// TIA Portal V20 export
FUNCTION_BLOCK "LER_StackLight"   // FB8, LAD
// stored: Access Published, MemoryReserve 100, SetENOAutomatically false
   VAR_INPUT
      stateDetail : "LER_typeStateDetail";
      powerOn : Bool;
      auto : Bool;
      manual : Bool;
   END_VAR
   VAR_OUTPUT
      setDone : Bool;
      signalStack : "LUC_typeSignalStackConfiguration";
   END_VAR
   VAR
      statExcute : Bool;
      statDefault : Bool;
      statReset : Bool;
      statResetDone : Bool;
      statPreStateDetail : "LER_typeStateDetail";
   END_VAR
   VAR_TEMP
      signalStackDelete : "LUC_typeSignalStackConfiguration";
      tempRetVal : Array[0..9] of Int;
   END_VAR
   VAR_TEMP   // added for the SCL form of the ladder/FBD networks
      _w1 : Bool;
   END_VAR
BEGIN

REGION Network 1 (SCL): stateDefault
   // stateDetail is All False
   IF (#stateDetail."Turn off" OR #stateDetail."Technical issue or alarm" OR #stateDetail."Internal starved" OR #stateDetail."Emergency or hazardous stop" OR #stateDetail.Overheat OR #stateDetail.Warning OR
       #stateDetail."External starved or blocked" OR #stateDetail."QC required soon" OR #stateDetail."Controlled Stop" OR #stateDetail."Ready to start" OR #stateDetail."Producing(running)") = 0 THEN
       #statDefault := TRUE;
       #statExcute := TRUE;
   END_IF;
END_REGION

REGION Network 2: reset
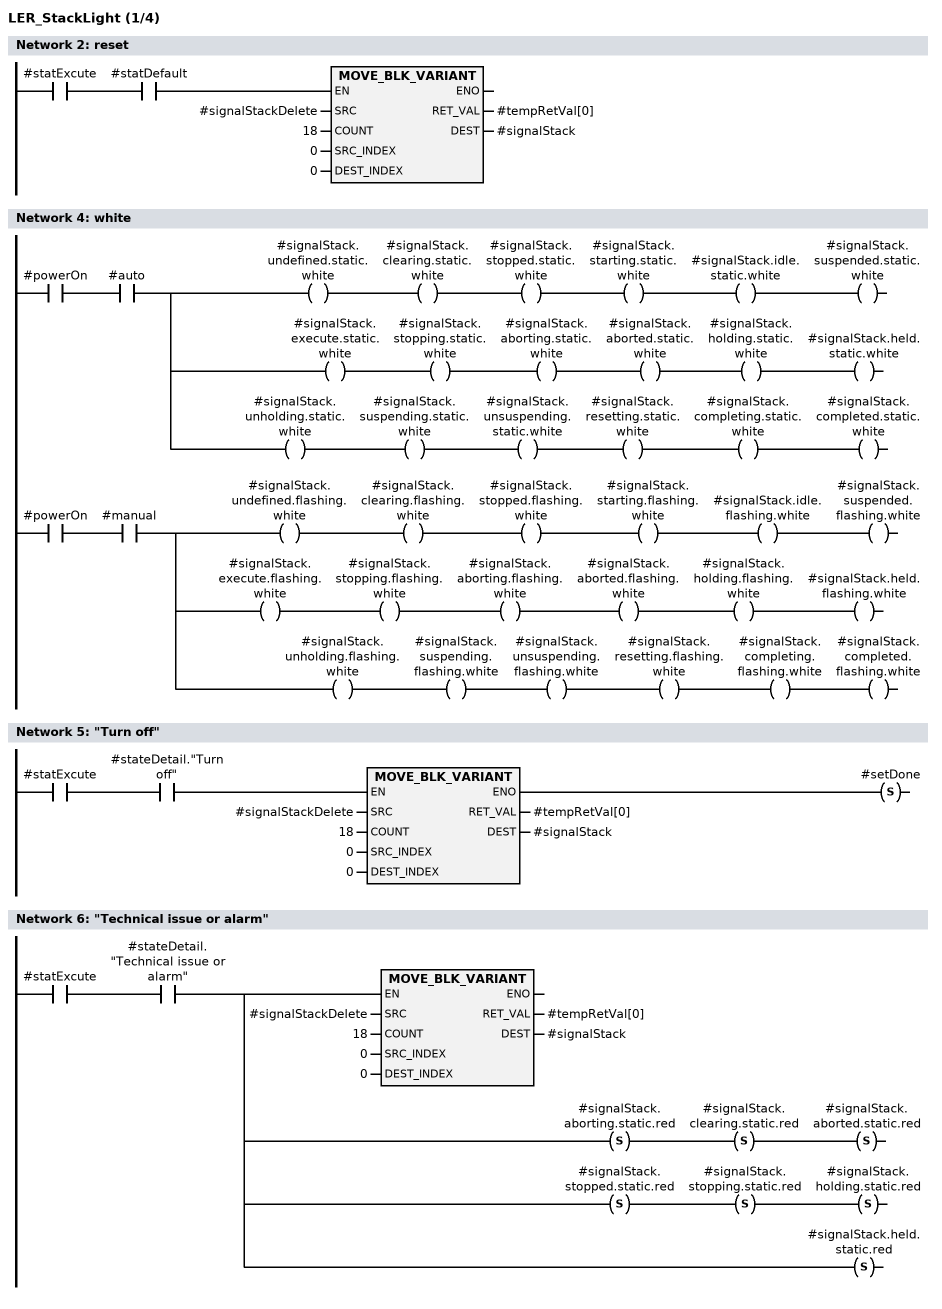
   RUNG wire#powerrail
      Contact( #statExcute )
      Contact( #statDefault )
      MOVE_BLK_VARIANT(SRC := #signalStackDelete, COUNT := 18, SRC_INDEX := 0, DEST_INDEX := 0, Ret_Val => #tempRetVal[0], DEST => #signalStack)
   END_RUNG
   // the same network as SCL:
   IF #statExcute AND #statDefault THEN
       #tempRetVal[0] := MOVE_BLK_VARIANT(SRC := #signalStackDelete,
                               COUNT := 18,
                               SRC_INDEX := 0,
                               DEST_INDEX := 0,
                               DEST => #signalStack);
   END_IF;
END_REGION

REGION Network 3 (SCL)
   IF #statPreStateDetail <> #stateDetail THEN
       #statExcute := TRUE;
       #statPreStateDetail := #stateDetail;
   END_IF;
END_REGION

REGION Network 4: white
   RUNG wire#powerrail
      Contact( #powerOn )
      Contact( #auto )
      wire#w1
      Coil( #signalStack.undefined.static.white )
      Coil( #signalStack.clearing.static.white )
      Coil( #signalStack.stopped.static.white )
      Coil( #signalStack.starting.static.white )
      Coil( #signalStack.idle.static.white )
      Coil( #signalStack.suspended.static.white )
   END_RUNG
   RUNG wire#w1
      Coil( #signalStack.execute.static.white )
      Coil( #signalStack.stopping.static.white )
      Coil( #signalStack.aborting.static.white )
      Coil( #signalStack.aborted.static.white )
      Coil( #signalStack.holding.static.white )
      Coil( #signalStack.held.static.white )
   END_RUNG
   RUNG wire#w1
      Coil( #signalStack.unholding.static.white )
      Coil( #signalStack.suspending.static.white )
      Coil( #signalStack.unsuspending.static.white )
      Coil( #signalStack.resetting.static.white )
      Coil( #signalStack.completing.static.white )
      Coil( #signalStack.completed.static.white )
   END_RUNG
   RUNG wire#powerrail
      Contact( #powerOn )
      Contact( #manual )
      wire#w2
      Coil( #signalStack.undefined.flashing.white )
      Coil( #signalStack.clearing.flashing.white )
      Coil( #signalStack.stopped.flashing.white )
      Coil( #signalStack.starting.flashing.white )
      Coil( #signalStack.idle.flashing.white )
      Coil( #signalStack.suspended.flashing.white )
   END_RUNG
   RUNG wire#w2
      Coil( #signalStack.execute.flashing.white )
      Coil( #signalStack.stopping.flashing.white )
      Coil( #signalStack.aborting.flashing.white )
      Coil( #signalStack.aborted.flashing.white )
      Coil( #signalStack.holding.flashing.white )
      Coil( #signalStack.held.flashing.white )
   END_RUNG
   RUNG wire#w2
      Coil( #signalStack.unholding.flashing.white )
      Coil( #signalStack.suspending.flashing.white )
      Coil( #signalStack.unsuspending.flashing.white )
      Coil( #signalStack.resetting.flashing.white )
      Coil( #signalStack.completing.flashing.white )
      Coil( #signalStack.completed.flashing.white )
   END_RUNG
   // the same network as SCL:
   #signalStack.undefined.static.white := #powerOn AND #auto;
   #signalStack.clearing.static.white := #signalStack.undefined.static.white;
   #signalStack.stopped.static.white := #signalStack.undefined.static.white;
   #signalStack.starting.static.white := #signalStack.undefined.static.white;
   #signalStack.idle.static.white := #signalStack.undefined.static.white;
   #signalStack.suspended.static.white := #signalStack.undefined.static.white;
   #signalStack.execute.static.white := #signalStack.undefined.static.white;
   #signalStack.stopping.static.white := #signalStack.undefined.static.white;
   #signalStack.aborting.static.white := #signalStack.undefined.static.white;
   #signalStack.aborted.static.white := #signalStack.undefined.static.white;
   #signalStack.holding.static.white := #signalStack.undefined.static.white;
   #signalStack.held.static.white := #signalStack.undefined.static.white;
   #signalStack.unholding.static.white := #signalStack.undefined.static.white;
   #signalStack.suspending.static.white := #signalStack.undefined.static.white;
   #signalStack.unsuspending.static.white := #signalStack.undefined.static.white;
   #signalStack.resetting.static.white := #signalStack.undefined.static.white;
   #signalStack.completing.static.white := #signalStack.undefined.static.white;
   #signalStack.completed.static.white := #signalStack.undefined.static.white;
   #signalStack.undefined.flashing.white := #powerOn AND #manual;
   #signalStack.clearing.flashing.white := #signalStack.undefined.flashing.white;
   #signalStack.stopped.flashing.white := #signalStack.undefined.flashing.white;
   #signalStack.starting.flashing.white := #signalStack.undefined.flashing.white;
   #signalStack.idle.flashing.white := #signalStack.undefined.flashing.white;
   #signalStack.suspended.flashing.white := #signalStack.undefined.flashing.white;
   #signalStack.execute.flashing.white := #signalStack.undefined.flashing.white;
   #signalStack.stopping.flashing.white := #signalStack.undefined.flashing.white;
   #signalStack.aborting.flashing.white := #signalStack.undefined.flashing.white;
   #signalStack.aborted.flashing.white := #signalStack.undefined.flashing.white;
   #signalStack.holding.flashing.white := #signalStack.undefined.flashing.white;
   #signalStack.held.flashing.white := #signalStack.undefined.flashing.white;
   #signalStack.unholding.flashing.white := #signalStack.undefined.flashing.white;
   #signalStack.suspending.flashing.white := #signalStack.undefined.flashing.white;
   #signalStack.unsuspending.flashing.white := #signalStack.undefined.flashing.white;
   #signalStack.resetting.flashing.white := #signalStack.undefined.flashing.white;
   #signalStack.completing.flashing.white := #signalStack.undefined.flashing.white;
   #signalStack.completed.flashing.white := #signalStack.undefined.flashing.white;
END_REGION

REGION Network 5: "Turn off"
   RUNG wire#powerrail
      Contact( #statExcute )
      Contact( #stateDetail."Turn off" )
      MOVE_BLK_VARIANT(SRC := #signalStackDelete, COUNT := 18, SRC_INDEX := 0, DEST_INDEX := 0, Ret_Val => #tempRetVal[0], DEST => #signalStack)
      S_Coil( #setDone )
   END_RUNG
   // the same network as SCL:
   #tempRetVal[0] := MOVE_BLK_VARIANT(EN := #statExcute AND #stateDetail."Turn off",
                           SRC := #signalStackDelete,
                           COUNT := 18,
                           SRC_INDEX := 0,
                           DEST_INDEX := 0,
                           DEST => #signalStack,
                           ENO => #_w1);
   IF #_w1 THEN #setDone := TRUE; END_IF;
END_REGION

REGION Network 6: "Technical issue or alarm"
   RUNG wire#powerrail
      Contact( #statExcute )
      Contact( #stateDetail."Technical issue or alarm" )
      wire#w1
      MOVE_BLK_VARIANT(SRC := #signalStackDelete, COUNT := 18, SRC_INDEX := 0, DEST_INDEX := 0, Ret_Val => #tempRetVal[0], DEST => #signalStack)
   END_RUNG
   RUNG wire#w1
      S_Coil( #signalStack.aborting.static.red )
      S_Coil( #signalStack.clearing.static.red )
      S_Coil( #signalStack.aborted.static.red )
   END_RUNG
   RUNG wire#w1
      S_Coil( #signalStack.stopped.static.red )
      S_Coil( #signalStack.stopping.static.red )
      S_Coil( #signalStack.holding.static.red )
   END_RUNG
   RUNG wire#w1
      S_Coil( #signalStack.held.static.red )
   END_RUNG
   // the same network as SCL:
   IF #statExcute AND #stateDetail."Technical issue or alarm" THEN
       #tempRetVal[0] := MOVE_BLK_VARIANT(SRC := #signalStackDelete,
                               COUNT := 18,
                               SRC_INDEX := 0,
                               DEST_INDEX := 0,
                               DEST => #signalStack);
       #signalStack.aborting.static.red := TRUE;
       #signalStack.clearing.static.red := TRUE;
       #signalStack.aborted.static.red := TRUE;
       #signalStack.stopped.static.red := TRUE;
       #signalStack.stopping.static.red := TRUE;
       #signalStack.holding.static.red := TRUE;
       #signalStack.held.static.red := TRUE;
   END_IF;
END_REGION

REGION Network 7: "Internal starved"
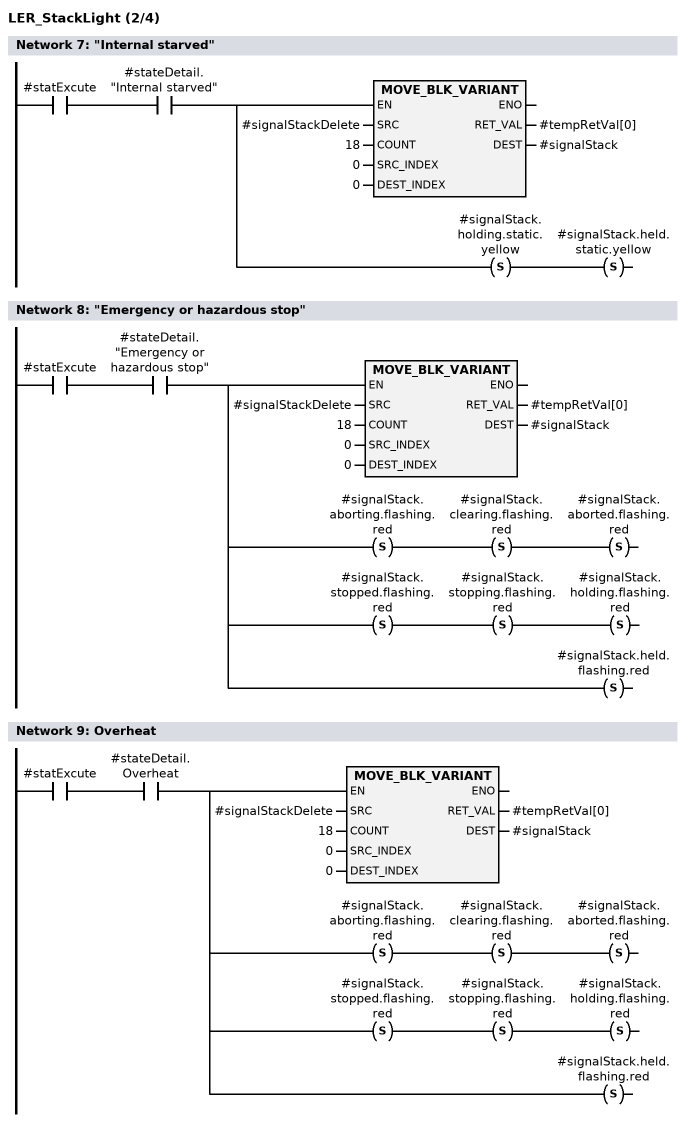
   RUNG wire#powerrail
      Contact( #statExcute )
      Contact( #stateDetail."Internal starved" )
      wire#w1
      MOVE_BLK_VARIANT(SRC := #signalStackDelete, COUNT := 18, SRC_INDEX := 0, DEST_INDEX := 0, Ret_Val => #tempRetVal[0], DEST => #signalStack)
   END_RUNG
   RUNG wire#w1
      S_Coil( #signalStack.holding.static.yellow )
      S_Coil( #signalStack.held.static.yellow )
   END_RUNG
   // the same network as SCL:
   IF #statExcute AND #stateDetail."Internal starved" THEN
       #tempRetVal[0] := MOVE_BLK_VARIANT(SRC := #signalStackDelete,
                               COUNT := 18,
                               SRC_INDEX := 0,
                               DEST_INDEX := 0,
                               DEST => #signalStack);
       #signalStack.holding.static.yellow := TRUE;
       #signalStack.held.static.yellow := TRUE;
   END_IF;
END_REGION

REGION Network 8: "Emergency or hazardous stop"
   RUNG wire#powerrail
      Contact( #statExcute )
      Contact( #stateDetail."Emergency or hazardous stop" )
      wire#w1
      MOVE_BLK_VARIANT(SRC := #signalStackDelete, COUNT := 18, SRC_INDEX := 0, DEST_INDEX := 0, Ret_Val => #tempRetVal[0], DEST => #signalStack)
   END_RUNG
   RUNG wire#w1
      S_Coil( #signalStack.aborting.flashing.red )
      S_Coil( #signalStack.clearing.flashing.red )
      S_Coil( #signalStack.aborted.flashing.red )
   END_RUNG
   RUNG wire#w1
      S_Coil( #signalStack.stopped.flashing.red )
      S_Coil( #signalStack.stopping.flashing.red )
      S_Coil( #signalStack.holding.flashing.red )
   END_RUNG
   RUNG wire#w1
      S_Coil( #signalStack.held.flashing.red )
   END_RUNG
   // the same network as SCL:
   IF #statExcute AND #stateDetail."Emergency or hazardous stop" THEN
       #tempRetVal[0] := MOVE_BLK_VARIANT(SRC := #signalStackDelete,
                               COUNT := 18,
                               SRC_INDEX := 0,
                               DEST_INDEX := 0,
                               DEST => #signalStack);
       #signalStack.aborting.flashing.red := TRUE;
       #signalStack.clearing.flashing.red := TRUE;
       #signalStack.aborted.flashing.red := TRUE;
       #signalStack.stopped.flashing.red := TRUE;
       #signalStack.stopping.flashing.red := TRUE;
       #signalStack.holding.flashing.red := TRUE;
       #signalStack.held.flashing.red := TRUE;
   END_IF;
END_REGION

REGION Network 9: Overheat
   RUNG wire#powerrail
      Contact( #statExcute )
      Contact( #stateDetail.Overheat )
      wire#w1
      MOVE_BLK_VARIANT(SRC := #signalStackDelete, COUNT := 18, SRC_INDEX := 0, DEST_INDEX := 0, Ret_Val => #tempRetVal[0], DEST => #signalStack)
   END_RUNG
   RUNG wire#w1
      S_Coil( #signalStack.aborting.flashing.red )
      S_Coil( #signalStack.clearing.flashing.red )
      S_Coil( #signalStack.aborted.flashing.red )
   END_RUNG
   RUNG wire#w1
      S_Coil( #signalStack.stopped.flashing.red )
      S_Coil( #signalStack.stopping.flashing.red )
      S_Coil( #signalStack.holding.flashing.red )
   END_RUNG
   RUNG wire#w1
      S_Coil( #signalStack.held.flashing.red )
   END_RUNG
   // the same network as SCL:
   IF #statExcute AND #stateDetail.Overheat THEN
       #tempRetVal[0] := MOVE_BLK_VARIANT(SRC := #signalStackDelete,
                               COUNT := 18,
                               SRC_INDEX := 0,
                               DEST_INDEX := 0,
                               DEST => #signalStack);
       #signalStack.aborting.flashing.red := TRUE;
       #signalStack.clearing.flashing.red := TRUE;
       #signalStack.aborted.flashing.red := TRUE;
       #signalStack.stopped.flashing.red := TRUE;
       #signalStack.stopping.flashing.red := TRUE;
       #signalStack.holding.flashing.red := TRUE;
       #signalStack.held.flashing.red := TRUE;
   END_IF;
END_REGION

REGION Network 10: Warning
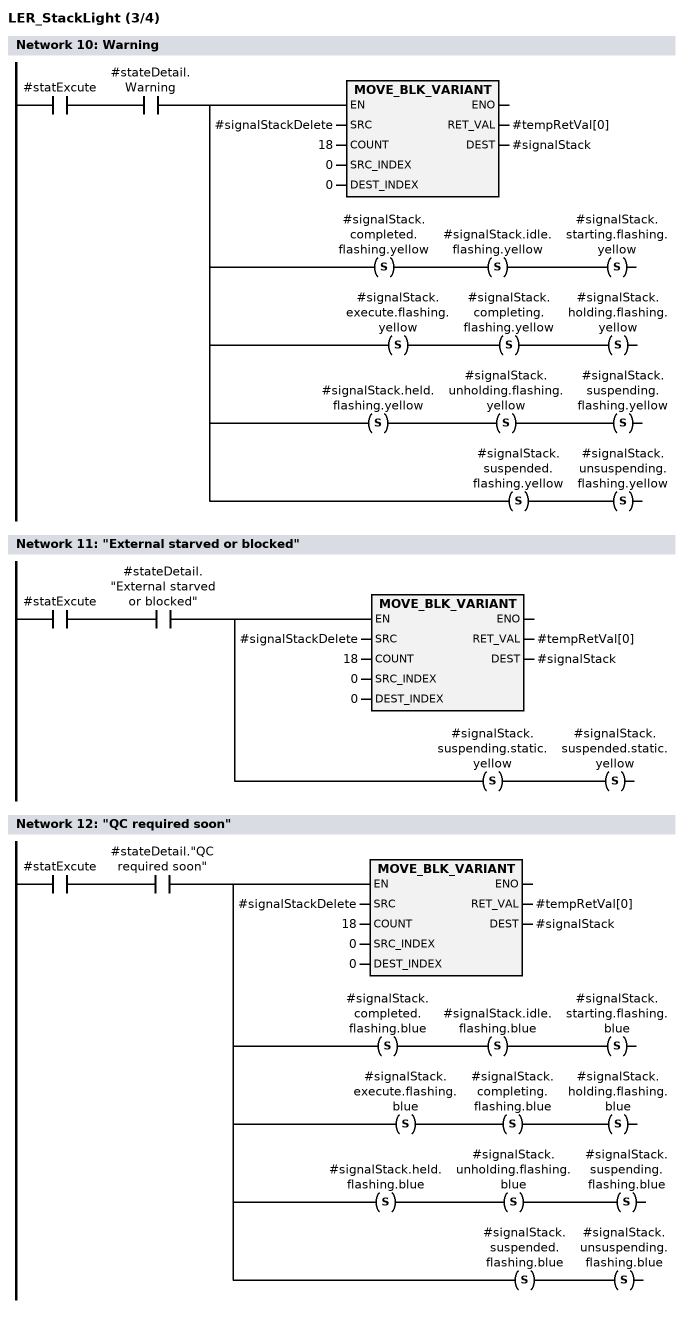
   RUNG wire#powerrail
      Contact( #statExcute )
      Contact( #stateDetail.Warning )
      wire#w1
      MOVE_BLK_VARIANT(SRC := #signalStackDelete, COUNT := 18, SRC_INDEX := 0, DEST_INDEX := 0, Ret_Val => #tempRetVal[0], DEST => #signalStack)
   END_RUNG
   RUNG wire#w1
      S_Coil( #signalStack.completed.flashing.yellow )
      S_Coil( #signalStack.idle.flashing.yellow )
      S_Coil( #signalStack.starting.flashing.yellow )
   END_RUNG
   RUNG wire#w1
      S_Coil( #signalStack.execute.flashing.yellow )
      S_Coil( #signalStack.completing.flashing.yellow )
      S_Coil( #signalStack.holding.flashing.yellow )
   END_RUNG
   RUNG wire#w1
      S_Coil( #signalStack.held.flashing.yellow )
      S_Coil( #signalStack.unholding.flashing.yellow )
      S_Coil( #signalStack.suspending.flashing.yellow )
   END_RUNG
   RUNG wire#w1
      S_Coil( #signalStack.suspended.flashing.yellow )
      S_Coil( #signalStack.unsuspending.flashing.yellow )
   END_RUNG
   // the same network as SCL:
   IF #statExcute AND #stateDetail.Warning THEN
       #tempRetVal[0] := MOVE_BLK_VARIANT(SRC := #signalStackDelete,
                               COUNT := 18,
                               SRC_INDEX := 0,
                               DEST_INDEX := 0,
                               DEST => #signalStack);
       #signalStack.completed.flashing.yellow := TRUE;
       #signalStack.idle.flashing.yellow := TRUE;
       #signalStack.starting.flashing.yellow := TRUE;
       #signalStack.execute.flashing.yellow := TRUE;
       #signalStack.completing.flashing.yellow := TRUE;
       #signalStack.holding.flashing.yellow := TRUE;
       #signalStack.held.flashing.yellow := TRUE;
       #signalStack.unholding.flashing.yellow := TRUE;
       #signalStack.suspending.flashing.yellow := TRUE;
       #signalStack.suspended.flashing.yellow := TRUE;
       #signalStack.unsuspending.flashing.yellow := TRUE;
   END_IF;
END_REGION

REGION Network 11: "External starved or blocked"
   RUNG wire#powerrail
      Contact( #statExcute )
      Contact( #stateDetail."External starved or blocked" )
      wire#w1
      MOVE_BLK_VARIANT(SRC := #signalStackDelete, COUNT := 18, SRC_INDEX := 0, DEST_INDEX := 0, Ret_Val => #tempRetVal[0], DEST => #signalStack)
   END_RUNG
   RUNG wire#w1
      S_Coil( #signalStack.suspending.static.yellow )
      S_Coil( #signalStack.suspended.static.yellow )
   END_RUNG
   // the same network as SCL:
   IF #statExcute AND #stateDetail."External starved or blocked" THEN
       #tempRetVal[0] := MOVE_BLK_VARIANT(SRC := #signalStackDelete,
                               COUNT := 18,
                               SRC_INDEX := 0,
                               DEST_INDEX := 0,
                               DEST => #signalStack);
       #signalStack.suspending.static.yellow := TRUE;
       #signalStack.suspended.static.yellow := TRUE;
   END_IF;
END_REGION

REGION Network 12: "QC required soon"
   RUNG wire#powerrail
      Contact( #statExcute )
      Contact( #stateDetail."QC required soon" )
      wire#w1
      MOVE_BLK_VARIANT(SRC := #signalStackDelete, COUNT := 18, SRC_INDEX := 0, DEST_INDEX := 0, Ret_Val => #tempRetVal[0], DEST => #signalStack)
   END_RUNG
   RUNG wire#w1
      S_Coil( #signalStack.completed.flashing.blue )
      S_Coil( #signalStack.idle.flashing.blue )
      S_Coil( #signalStack.starting.flashing.blue )
   END_RUNG
   RUNG wire#w1
      S_Coil( #signalStack.execute.flashing.blue )
      S_Coil( #signalStack.completing.flashing.blue )
      S_Coil( #signalStack.holding.flashing.blue )
   END_RUNG
   RUNG wire#w1
      S_Coil( #signalStack.held.flashing.blue )
      S_Coil( #signalStack.unholding.flashing.blue )
      S_Coil( #signalStack.suspending.flashing.blue )
   END_RUNG
   RUNG wire#w1
      S_Coil( #signalStack.suspended.flashing.blue )
      S_Coil( #signalStack.unsuspending.flashing.blue )
   END_RUNG
   // the same network as SCL:
   IF #statExcute AND #stateDetail."QC required soon" THEN
       #tempRetVal[0] := MOVE_BLK_VARIANT(SRC := #signalStackDelete,
                               COUNT := 18,
                               SRC_INDEX := 0,
                               DEST_INDEX := 0,
                               DEST => #signalStack);
       #signalStack.completed.flashing.blue := TRUE;
       #signalStack.idle.flashing.blue := TRUE;
       #signalStack.starting.flashing.blue := TRUE;
       #signalStack.execute.flashing.blue := TRUE;
       #signalStack.completing.flashing.blue := TRUE;
       #signalStack.holding.flashing.blue := TRUE;
       #signalStack.held.flashing.blue := TRUE;
       #signalStack.unholding.flashing.blue := TRUE;
       #signalStack.suspending.flashing.blue := TRUE;
       #signalStack.suspended.flashing.blue := TRUE;
       #signalStack.unsuspending.flashing.blue := TRUE;
   END_IF;
END_REGION

REGION Network 13: "Controlled Stop"
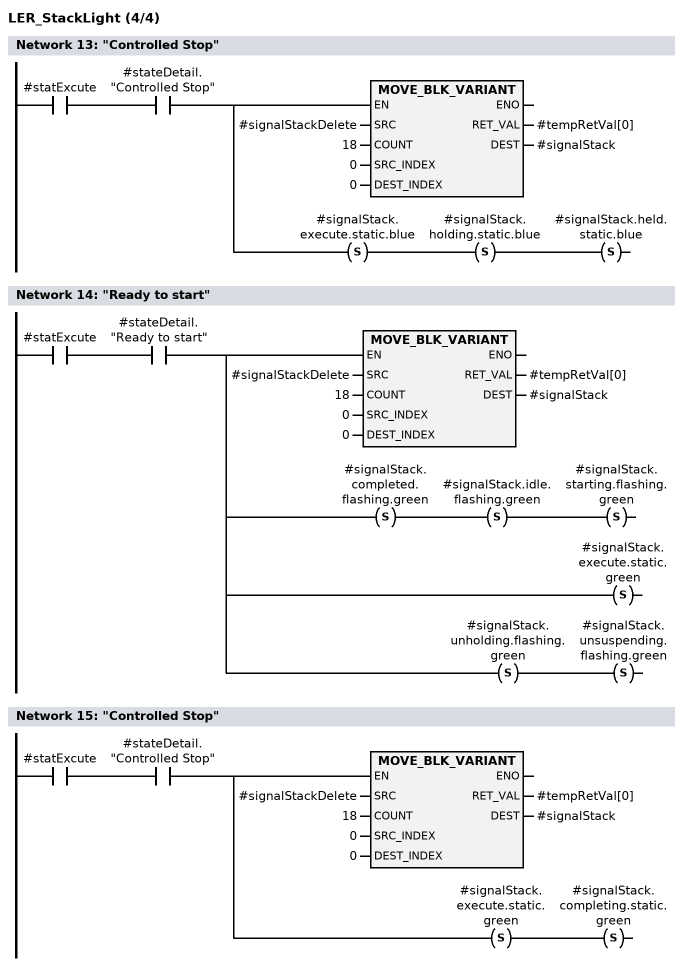
   RUNG wire#powerrail
      Contact( #statExcute )
      Contact( #stateDetail."Controlled Stop" )
      wire#w1
      MOVE_BLK_VARIANT(SRC := #signalStackDelete, COUNT := 18, SRC_INDEX := 0, DEST_INDEX := 0, Ret_Val => #tempRetVal[0], DEST => #signalStack)
   END_RUNG
   RUNG wire#w1
      S_Coil( #signalStack.execute.static.blue )
      S_Coil( #signalStack.holding.static.blue )
      S_Coil( #signalStack.held.static.blue )
   END_RUNG
   // the same network as SCL:
   IF #statExcute AND #stateDetail."Controlled Stop" THEN
       #tempRetVal[0] := MOVE_BLK_VARIANT(SRC := #signalStackDelete,
                               COUNT := 18,
                               SRC_INDEX := 0,
                               DEST_INDEX := 0,
                               DEST => #signalStack);
       #signalStack.execute.static.blue := TRUE;
       #signalStack.holding.static.blue := TRUE;
       #signalStack.held.static.blue := TRUE;
   END_IF;
END_REGION

REGION Network 14: "Ready to start"
   RUNG wire#powerrail
      Contact( #statExcute )
      Contact( #stateDetail."Ready to start" )
      wire#w1
      MOVE_BLK_VARIANT(SRC := #signalStackDelete, COUNT := 18, SRC_INDEX := 0, DEST_INDEX := 0, Ret_Val => #tempRetVal[0], DEST => #signalStack)
   END_RUNG
   RUNG wire#w1
      S_Coil( #signalStack.completed.flashing.green )
      S_Coil( #signalStack.idle.flashing.green )
      S_Coil( #signalStack.starting.flashing.green )
   END_RUNG
   RUNG wire#w1
      S_Coil( #signalStack.execute.static.green )
   END_RUNG
   RUNG wire#w1
      S_Coil( #signalStack.unholding.flashing.green )
      S_Coil( #signalStack.unsuspending.flashing.green )
   END_RUNG
   // the same network as SCL:
   IF #statExcute AND #stateDetail."Ready to start" THEN
       #tempRetVal[0] := MOVE_BLK_VARIANT(SRC := #signalStackDelete,
                               COUNT := 18,
                               SRC_INDEX := 0,
                               DEST_INDEX := 0,
                               DEST => #signalStack);
       #signalStack.completed.flashing.green := TRUE;
       #signalStack.idle.flashing.green := TRUE;
       #signalStack.starting.flashing.green := TRUE;
       #signalStack.execute.static.green := TRUE;
       #signalStack.unholding.flashing.green := TRUE;
       #signalStack.unsuspending.flashing.green := TRUE;
   END_IF;
END_REGION

REGION Network 15: "Controlled Stop"
   RUNG wire#powerrail
      Contact( #statExcute )
      Contact( #stateDetail."Controlled Stop" )
      wire#w1
      MOVE_BLK_VARIANT(SRC := #signalStackDelete, COUNT := 18, SRC_INDEX := 0, DEST_INDEX := 0, Ret_Val => #tempRetVal[0], DEST => #signalStack)
   END_RUNG
   RUNG wire#w1
      S_Coil( #signalStack.execute.static.green )
      S_Coil( #signalStack.completing.static.green )
   END_RUNG
   // the same network as SCL:
   IF #statExcute AND #stateDetail."Controlled Stop" THEN
       #tempRetVal[0] := MOVE_BLK_VARIANT(SRC := #signalStackDelete,
                               COUNT := 18,
                               SRC_INDEX := 0,
                               DEST_INDEX := 0,
                               DEST => #signalStack);
       #signalStack.execute.static.green := TRUE;
       #signalStack.completing.static.green := TRUE;
   END_IF;
END_REGION
END_FUNCTION_BLOCK
